PROGRAM readTemp
VAR
	fbRecGeneric		: 	FB_Rec_Generic;
END_VAR
VAR_INPUT
	sensorID			: DWORD;
END_VAR
VAR_OUTPUT
	tempOutput			: LREAL;
	humitityOut			: LREAL;
END_VAR

fbRecGeneric(str_KL6581 := GVL_EnOcean.stKL6581, byNode := 0, dw_ID := sensorID);

IF fbRecGeneric.bReceive = FALSE THEN
	tempOutput := F_Scale(fRawData := fbRecGeneric.ar_Value[1], fRawDataLowerOffLimit := 0, fRawDataUpperOffLimit := 255, fScaleDataLowerOffLimit := -20, fScaleDataUpperOffLimit := 60);
	humitityOut := F_Scale(fRawData := fbRecGeneric.ar_Value[2], fRawDataLowerOffLimit := 0, fRawDataUpperOffLimit := 255, fScaleDataLowerOffLimit := 0, fScaleDataUpperOffLimit := 100);
	
	
END_IF

END_PROGRAM

(* stored: Version 1.1.0.1, ProductVersion 3.1.4022.17
   POU readTemp: Id {a05587da-b532-45bc-a256-2d989c37bb2a}, SpecialFunc None *)
